# B&R Automation Studio project CombinedLinenSoiledA9KAN (part 12)

```iecst
						_PmIntern.enCycImpState := cs_ImpRdyFault;

					ELSE

						_PmIntern.enCycImpState := cs_ImpTOC;

					END_IF

				END_IF

			cs_ImpDelDir:

				_DirDeleteEx(enable := TRUE, pDevice := ADR(KG_DEVICE_COMPACTFLASH), pName := ADR(_PmIntern.sActPath));

				IF _DirDeleteEx.status <> ERR_FUB_BUSY THEN

					_PmIntern.enCycImpState := cs_ImpTOC;

				END_IF

			cs_ImpTOC:

				_PmIntern.ExpSettings.sCfDeviceName := KG_DEVICE_COMPACTFLASH;
				_PmIntern.ExpSettings.sPath := MNPARAM_PATH_EXPORT;

				_ExportTableOfContent(Enable := TRUE, pIntern := ADR(_PmIntern));

				IF _ExportTableOfContent.Status = ERR_OK THEN

					mnParamStatAd.dtExportContent := _ExportTableOfContent.dtTocWritten;

					_PmIntern.enCycImpState := cs_ImpRdySuccess;

				ELSIF _ExportTableOfContent.Status <> ERR_FUB_BUSY THEN

					_PmIntern.Status.wMsgClass := 10;
					_PmIntern.Status.wMsgNumber := MNPARAM_MSG_WARN_IMPORT;
					_PmIntern.Status.diMsgAttr1 := _ExportTableOfContent.Status;
					_PmIntern.Status.diMsgAttr2 := _ExportTableOfContent.AdStatus;
					_PmIntern.Status.wMsgAckLevel := 0;

					_PmIntern.enCycImpState := cs_ImpRdyFault;

				END_IF

			cs_ImpRdyFault:

			// Mit Fehler beendet

			cs_ImpRdySuccess:

				// Mit Erfolg beendet

		END_CASE

		//*********************************************************************************************
		// Statemachine zum Füllen des Editiors mit Daten
		//*********************************************************************************************

		CASE _PmIntern.enCycFillEditor OF

			cs_feIdle:

			cs_feStart:

				brsmemset(ADR(IFmnParam.Out.Edit.AttrNum), 0, SIZEOF(IFmnParam.Out.Edit.AttrNum));
				brsmemset(ADR(IFmnParam.Out.Edit.AttrStr), 0, SIZEOF(IFmnParam.Out.Edit.AttrStr));
				IFmnParam.Out.Edit.bCntNumRows := 0;
				IFmnParam.Out.Edit.bCntStrRows := 0;
				IFmnParam.Out.Edit.bContainer := 0;
				IFmnParam.Out.Edit.wContainerInstance := 0;
				IFmnParam.Out.Edit.wRowNumOffset := 0;
				IFmnParam.Out.Edit.wRowStrOffset := 0;

				brsmemset(ADR(_EditNumValues), 0, SIZEOF(_EditNumValues));
				brsmemset(ADR(_EditStrValues), 0, SIZEOF(_EditStrValues));

				IFmnParam.Out.Edit.wStatus := KG_STAT_BUSY;

				_DefineActContainer(Enable := TRUE, bContainerIdx := IFmnParam.In.Edit.bContainer, wInstanceIdx := IFmnParam.In.Edit.wContainerInstance, pIntern := ADR(_PmIntern));

				IF _DefineActContainer.Status = ERR_OK THEN

					// Container Parameter sind im gültigen Bereich und die Containerspec. ist ok

					IF (_PmIntern.TOC.TocEntry[_PmIntern.TOC.wStartIdx[IFmnParam.In.Edit.bContainer] + (IFmnParam.In.Edit.wContainerInstance - _PmIntern.ActContainer.wMinBound)].xExist
						AND _PmIntern.ActContainer.bDirect = 0)
						OR
						(_PmIntern.TOC.TocEntry[_PmIntern.TOC.wStartIdx[IFmnParam.In.Edit.bContainer]].xExist AND _PmIntern.ActContainer.bDirect = 1) THEN

						// Die Containerinstanz existiert

						_diCSVNum(enable := TRUE, pName := ADR(_PmIntern.ActContainer.sDoNameNum));

						IF _diCSVNum.status = ERR_OK THEN

							// Datenobjekt mit aktuellen numerischen Parametern wurde gefunden

							_PmIntern.CSVDataObjects.Adress.lCSVNum := _diCSVNum.pDatObjMem;
							_PmIntern.CSVDataObjects.Size.lCSVNum := _diCSVNum.len;
							_PmIntern.CSVDataObjects.Idents.lCSVNum := _diCSVNum.ident;

							_pDoContainerNum ACCESS _PmIntern.CSVDataObjects.Adress.lCSVNum;

							_PmIntern.CSVDataObjects.MaxIndex.lCSVNum := ( (_pDoContainerNum.Header.Do.lActEndPos - SIZEOF(mnParam_CsvDynHeader_typ)) / SIZEOF(_pDoContainerNum.CsvNum[1]) );

							_diCSVString(enable := TRUE, pName := ADR(_PmIntern.ActContainer.sDoNameString));

							IF _diCSVString.status = ERR_OK THEN

								// Datenobjekt mit aktuellen String Parametern wurde gefunden

								_PmIntern.CSVDataObjects.Adress.lCSVString := _diCSVString.pDatObjMem;
								_PmIntern.CSVDataObjects.Size.lCSVString := _diCSVString.len;
								_PmIntern.CSVDataObjects.Idents.lCSVString := _diCSVString.ident;

								_pDoContainerString ACCESS _PmIntern.CSVDataObjects.Adress.lCSVString;

								_PmIntern.CSVDataObjects.MaxIndex.lCSVString := ( (_pDoContainerString.Header.Do.lActEndPos - SIZEOF(mnParam_CsvDynHeader_typ)) / SIZEOF(_pDoContainerString.CsvString[1]) );

								_PmIntern.enCycFillEditor := cs_feFillEditor;

							ELSIF _diCSVString.status <> ERR_FUB_BUSY THEN

								_PmIntern.Status.wMsgClass := 10;
								_PmIntern.Status.wMsgNumber := MNPARAM_MSG_WARN_FILLEDITOR;
								_PmIntern.Status.diMsgAttr1 := MNPARAM_STAT_SYSERROR;
								_PmIntern.Status.diMsgAttr2 := 0;
								_PmIntern.Status.sMsgAttrTxt := _PmIntern.ActContainer.sDoNameString;
								_PmIntern.Status.wMsgAckLevel := 0;

								_PmIntern.enCycFillEditor := cs_feRdyFault;

							END_IF

						ELSIF _diCSVNum.status <> ERR_FUB_BUSY THEN

							_PmIntern.Status.wMsgClass := 10;
							_PmIntern.Status.wMsgNumber := MNPARAM_MSG_WARN_FILLEDITOR;
							_PmIntern.Status.diMsgAttr1 := MNPARAM_STAT_SYSERROR;
							_PmIntern.Status.diMsgAttr2 := 0;
							_PmIntern.Status.sMsgAttrTxt := _PmIntern.ActContainer.sDoNameNum;
							_PmIntern.Status.wMsgAckLevel := 0;

							_PmIntern.enCycFillEditor := cs_feRdyFault;

						END_IF

					ELSE

						_PmIntern.Status.wMsgClass := 10;
						_PmIntern.Status.wMsgNumber := MNPARAM_MSG_WARN_FILLEDITOR;
						_PmIntern.Status.diMsgAttr1 := MNPARAM_STAT_CONTINST_NOT_EXIST;
						_PmIntern.Status.diMsgAttr2 := 0;
						_PmIntern.Status.wMsgAckLevel := 0;

						_PmIntern.enCycFillEditor := cs_feRdyFault;

					END_IF

				ELSE

					_PmIntern.Status.wMsgClass := 10;
					_PmIntern.Status.wMsgNumber := MNPARAM_MSG_WARN_FILLEDITOR;
					_PmIntern.Status.diMsgAttr1 := _DefineActContainer.Status;
					_PmIntern.Status.diMsgAttr2 := 0;
					_PmIntern.Status.wMsgAckLevel := 0;

					_PmIntern.enCycFillEditor := cs_feRdyFault;

				END_IF

			cs_feFillEditor:

				IFmnParam.Out.Edit.bContainer := IFmnParam.In.Edit.bContainer;
				IFmnParam.Out.Edit.wContainerInstance := IFmnParam.In.Edit.wContainerInstance;
				IFmnParam.Out.Edit.wRowStrOffset := IFmnParam.In.Edit.wRowStrOffset;
				IFmnParam.Out.Edit.lPtrEditNumValues := ADR(_EditNumValues);
				IFmnParam.Out.Edit.lPtrEditStrValues := ADR(_EditStrValues);

				// Numerische Werte auslesen

				IF _PmIntern.CSVDataObjects.MaxIndex.lCSVNum > 0 AND IFmnParam.In.Edit.bCntNumRows > 0 THEN

					IF IFmnParam.In.Edit.bSelectModeNum = MNPARAM_SELECTMODE_LINEAR THEN

						IFmnParam.Out.Edit.wRowNumOffset := IFmnParam.In.Edit.wRowNumOffset;
						_wActRow := 1;
						_wActIdx := 1 + IFmnParam.In.Edit.wRowNumOffset;;

						REPEAT

							// Nur ausführen, wenn _wActIdx zulässig ist
							IF _wActIdx <= _PmIntern.CSVDataObjects.MaxIndex.lCSVNum THEN

								// Referenz auf Parameterbeschreibung auslesen
								_wActRefIdx := _pDoContainerNum.CsvNum[_wActIdx].wIdxNumPar;

								// Ist die Referenz zulässig, d.h. ist der Parameter im Modell definiert?
								IF _wActRefIdx <= _PmIntern.DataObjects.MaxIndex.lParamNum THEN

									// Schreib- und Leserechte ermitteln. Sie können vererbt sein!
									_GetAccessRights(Enable := TRUE, siWriteAccess := _pDoParamNum.ParamNum[_wActRefIdx].siWriteAccess,
										siReadAccess := _pDoParamNum.ParamNum[_wActRefIdx].siVisibleAccess,
										wReference := _pDoParamNum.ParamNum[_wActRefIdx].wReferenz,
										lPtrLogicStruct := _PmIntern.DataObjects.Adress.lLogicalStruct,
										wMaxIdxLogicStruct := UDINT_TO_UINT(_PmIntern.DataObjects.MaxIndex.lLogicalStruct));

									IF _GetAccessRights.bReadAccess <= IFmnParam.In.Edit.bUserLevel THEN

										IFmnParam.Out.Edit.AttrNum[_wActRow].bReadAccess := _GetAccessRights.bReadAccess;
										IFmnParam.Out.Edit.AttrNum[_wActRow].bWriteAccess := _GetAccessRights.bWriteAccess;

										// ***************ACTION***************
										_actFillEditNum;
										// ***************ACTION***************

										IFmnParam.Out.Edit.bCntNumRows := UINT_TO_USINT(_wActRow);

										_wActRow := _wActRow + 1;

									END_IF

								END_IF

							END_IF

							_wActIdx := _wActIdx + 1;

							UNTIL

							_PmIntern.CSVDataObjects.MaxIndex.lCSVNum < _wActIdx OR _wActRow > MIN(MNPARAM_CNT_EDITROWS, IFmnParam.In.Edit.bCntNumRows)

						END_REPEAT

					// Stringwerte auslesen, wenn gefordert

					ELSIF IFmnParam.In.Edit.bSelectModeNum = MNPARAM_SELECTMODE_BYIDX THEN

						IFmnParam.Out.Edit.wRowNumOffset := 0;
						IFmnParam.Out.Edit.bCntNumRows := UINT_TO_USINT(MIN(MNPARAM_CNT_EDITROWS, IFmnParam.In.Edit.bCntNumRows));

						FOR _ii := 1 TO IFmnParam.Out.Edit.bCntNumRows DO

							_wActRow := _ii;

							// Ist die Referenz zulässig, d.h. ist der Parameter im Modell definiert?
							IF IFmnParam.In.Edit.wSelParIdxNum[_wActRow] <= _PmIntern.DataObjects.MaxIndex.lParamNum AND IFmnParam.In.Edit.wSelParIdxNum[_wActRow] > 0 THEN

								_wActRefIdx := IFmnParam.In.Edit.wSelParIdxNum[_wActRow];

								// Suche Parameter-Containerindex anhand des Parameterindex und der 4 möglichen Array-Werte
								_binarySearchNum.enable := TRUE;
								_binarySearchNum.CsvStructNum.wIdxNumPar 	:= IFmnParam.In.Edit.wSelParIdxNum[_wActRow];
								_binarySearchNum.CsvStructNum.wArrIdx1 		:= IFmnParam.In.Edit.wSelParArrIdxNum[_wActRow,1];
								_binarySearchNum.CsvStructNum.wArrIdx2 		:= IFmnParam.In.Edit.wSelParArrIdxNum[_wActRow,2];
								_binarySearchNum.CsvStructNum.wArrIdx3 		:= IFmnParam.In.Edit.wSelParArrIdxNum[_wActRow,3];
								_binarySearchNum.CsvStructNum.wArrIdx4 		:= IFmnParam.In.Edit.wSelParArrIdxNum[_wActRow,4];
								_binarySearchNum.lpList 					:= _PmIntern.CSVDataObjects.Adress.lCSVNum;
								_binarySearchNum.lMaxRow 					:= _PmIntern.CSVDataObjects.MaxIndex.lCSVNum;

								_binarySearchNum();

								// Wurde der Parameter im Container gefunden ?
								IF _binarySearchNum.status = ERR_OK THEN

									_wActIdx := UDINT_TO_UINT(_binarySearchNum.lFoundRow);

									// Schreib- und Leserechte ermitteln. Sie können vererbt sein!
									_GetAccessRights(Enable := TRUE, siWriteAccess := _pDoParamNum.ParamNum[_wActRefIdx].siWriteAccess,
										siReadAccess := _pDoParamNum.ParamNum[_wActRefIdx].siVisibleAccess,
										wReference := _pDoParamNum.ParamNum[_wActRefIdx].wReferenz,
										lPtrLogicStruct := _PmIntern.DataObjects.Adress.lLogicalStruct,
										wMaxIdxLogicStruct := UDINT_TO_UINT(_PmIntern.DataObjects.MaxIndex.lLogicalStruct));

									IF _GetAccessRights.bReadAccess <= IFmnParam.In.Edit.bUserLevel THEN

										IFmnParam.Out.Edit.AttrNum[_wActRow].bReadAccess := _GetAccessRights.bReadAccess;
										IFmnParam.Out.Edit.AttrNum[_wActRow].bWriteAccess := _GetAccessRights.bWriteAccess;

										// ***************ACTION***************
										_actFillEditNum;
										// ***************ACTION***************

									END_IF

								END_IF

							END_IF

						END_FOR

					END_IF

				END_IF

				IF _PmIntern.CSVDataObjects.MaxIndex.lCSVString > 0 AND IFmnParam.In.Edit.bCntStrRows > 0 THEN

					IF IFmnParam.In.Edit.bSelectModeStr = MNPARAM_SELECTMODE_LINEAR THEN

						IFmnParam.Out.Edit.wRowStrOffset := IFmnParam.In.Edit.wRowStrOffset;
						_wActRow := 1;
						_wActIdx := 1 + IFmnParam.In.Edit.wRowStrOffset;;

						REPEAT

							// Nur ausführen, wenn _wActIdx zulässig ist
							IF _wActIdx <= _PmIntern.CSVDataObjects.MaxIndex.lCSVString THEN

								// Referenz auf Parameterbeschreibung auslesen
								_wActRefIdx := _pDoContainerString.CsvString[_wActIdx].wIdxStringPar;

								// Ist die Referenz zulässig, d.h. ist der Parameter im Modell definiert?
								IF _wActRefIdx <= _PmIntern.DataObjects.MaxIndex.lParamString THEN

									// Schreib- und Leserechte ermitteln. Sie können vererbt sein!
									_GetAccessRights(Enable := TRUE, siWriteAccess := _pDoParamString.ParamString[_wActRefIdx].siWriteAccess,
									siReadAccess := _pDoParamString.ParamString[_wActRefIdx].siVisibleAccess,
									wReference := _pDoParamString.ParamString[_wActRefIdx].wReferenz,
									lPtrLogicStruct := _PmIntern.DataObjects.Adress.lLogicalStruct,
									wMaxIdxLogicStruct := UDINT_TO_UINT(_PmIntern.DataObjects.MaxIndex.lLogicalStruct));

									IF _GetAccessRights.bReadAccess <= IFmnParam.In.Edit.bUserLevel THEN

										IFmnParam.Out.Edit.AttrStr[_wActRow].bReadAccess := _GetAccessRights.bReadAccess;
										IFmnParam.Out.Edit.AttrStr[_wActRow].bWriteAccess := _GetAccessRights.bWriteAccess;

										// ***************ACTION***************
										_actFillEditStr;
										// ***************ACTION***************

										IFmnParam.Out.Edit.bCntStrRows := UINT_TO_USINT(_wActRow);

										_wActRow := _wActRow + 1;

									END_IF

								END_IF

							END_IF

							_wActIdx := _wActIdx + 1;

							UNTIL

							_PmIntern.CSVDataObjects.MaxIndex.lCSVString < _wActIdx OR _wActRow > MIN(MNPARAM_CNT_EDITROWS, IFmnParam.In.Edit.bCntStrRows)

						END_REPEAT

					ELSIF IFmnParam.In.Edit.bSelectModeStr = MNPARAM_SELECTMODE_BYIDX THEN

						IFmnParam.Out.Edit.wRowStrOffset := 0;
						IFmnParam.Out.Edit.bCntStrRows := UINT_TO_USINT(MIN(MNPARAM_CNT_EDITROWS, IFmnParam.In.Edit.bCntStrRows));

						FOR _ii := 1 TO IFmnParam.Out.Edit.bCntStrRows DO

							_wActRow := _ii;

							// Ist die Referenz zulässig, d.h. ist der Parameter im Modell definiert?
							IF IFmnParam.In.Edit.wSelParIdxStr[_wActRow] <= _PmIntern.DataObjects.MaxIndex.lParamString AND IFmnParam.In.Edit.wSelParIdxStr[_wActRow] > 0 THEN

								_wActRefIdx := IFmnParam.In.Edit.wSelParIdxStr[_wActRow];

								// Suche Parameter-Containerindex anhand des Parameterindex und der 4 möglichen Array-Werte
								_binarySearchString.enable := TRUE;
								_binarySearchString.CsvStructString.wIdxStringPar 	:= IFmnParam.In.Edit.wSelParIdxStr[_wActRow];
								_binarySearchString.CsvStructString.wArrIdx1 		:= IFmnParam.In.Edit.wSelParArrIdxStr[_wActRow,1];
								_binarySearchString.CsvStructString.wArrIdx2 		:= IFmnParam.In.Edit.wSelParArrIdxStr[_wActRow,2];
								_binarySearchString.CsvStructString.wArrIdx3 		:= IFmnParam.In.Edit.wSelParArrIdxStr[_wActRow,3];
								_binarySearchString.CsvStructString.wArrIdx4 		:= IFmnParam.In.Edit.wSelParArrIdxStr[_wActRow,4];
								_binarySearchString.lpList 							:= _PmIntern.CSVDataObjects.Adress.lCSVString;
								_binarySearchString.lMaxRow 						:= _PmIntern.CSVDataObjects.MaxIndex.lCSVString;

								_binarySearchString();

								// Wurde der Parameter im Container gefunden ?
								IF _binarySearchString.status = ERR_OK THEN

									_wActIdx := UDINT_TO_UINT(_binarySearchString.lFoundRow);

									// Schreib- und Leserechte ermitteln. Sie können vererbt sein!
									_GetAccessRights(Enable := TRUE, siWriteAccess := _pDoParamString.ParamString[_wActRefIdx].siWriteAccess,
									siReadAccess := _pDoParamString.ParamString[_wActRefIdx].siVisibleAccess,
									wReference := _pDoParamString.ParamString[_wActRefIdx].wReferenz,
									lPtrLogicStruct := _PmIntern.DataObjects.Adress.lLogicalStruct,
									wMaxIdxLogicStruct := UDINT_TO_UINT(_PmIntern.DataObjects.MaxIndex.lLogicalStruct));

									IF _GetAccessRights.bReadAccess <= IFmnParam.In.Edit.bUserLevel THEN

										IFmnParam.Out.Edit.AttrStr[_wActRow].bReadAccess := _GetAccessRights.bReadAccess;
										IFmnParam.Out.Edit.AttrStr[_wActRow].bWriteAccess := _GetAccessRights.bWriteAccess;

										// ***************ACTION***************
										_actFillEditStr;
										// ***************ACTION***************

									END_IF

								END_IF

							END_IF

						END_FOR

					END_IF

				END_IF

				_PmIntern.enCycFillEditor := cs_feRdySuccess;

			cs_feRdyFault:

			// Mit Fehler beendet

			cs_feRdySuccess:

				// Erfolgreich beendet

		END_CASE

		//*********************************************************************************************
		// Statemachine zum Sichern der Daten des Editiors
		//*********************************************************************************************

		CASE _PmIntern.enCycSaveEditor OF

			cs_seIdle:

			cs_seStart:

				_DefineActContainer(Enable := TRUE, bContainerIdx := IFmnParam.In.Edit.bContainer, wInstanceIdx := IFmnParam.In.Edit.wContainerInstance, pIntern := ADR(_PmIntern));

				IF _DefineActContainer.Status = ERR_OK THEN

					// Container Parameter sind im gültigen Bereich und die Containerspec. ist ok

					IF 	(_PmIntern.TOC.TocEntry[_PmIntern.TOC.wStartIdx[IFmnParam.In.Edit.bContainer] + (IFmnParam.In.Edit.wContainerInstance - _PmIntern.ActContainer.wMinBound)].xExist
						AND _PmIntern.ActContainer.bDirect = 0)
						OR
						(_PmIntern.TOC.TocEntry[_PmIntern.TOC.wStartIdx[IFmnParam.In.Edit.bContainer]].xExist AND _PmIntern.ActContainer.bDirect = 1) THEN

						// Die Containerinstanz existiert

						_diCSVNum(enable := TRUE, pName := ADR(_PmIntern.ActContainer.sDoNameNum));

						IF _diCSVNum.status = ERR_OK THEN

							// Datenobjekt mit aktuellen numerischen Parametern wurde gefunden

							_PmIntern.CSVDataObjects.Adress.lCSVNum := _diCSVNum.pDatObjMem;
							_PmIntern.CSVDataObjects.Size.lCSVNum := _diCSVNum.len;
							_PmIntern.CSVDataObjects.Idents.lCSVNum := _diCSVNum.ident;

							_pDoContainerNum ACCESS _PmIntern.CSVDataObjects.Adress.lCSVNum;

							IF NOT _pDoContainerNum.Header.Container.xWriteProtected THEN

								_PmIntern.CSVDataObjects.MaxIndex.lCSVNum := ( (_pDoContainerNum.Header.Do.lActEndPos - SIZEOF(mnParam_CsvDynHeader_typ)) / SIZEOF(_pDoContainerNum.CsvNum[1]) );

								_diCSVString(enable := TRUE, pName := ADR(_PmIntern.ActContainer.sDoNameString));

								IF _diCSVString.status = ERR_OK THEN

									// Datenobjekt mit aktuellen String Parametern wurde gefunden

									_PmIntern.CSVDataObjects.Adress.lCSVString := _diCSVString.pDatObjMem;
									_PmIntern.CSVDataObjects.Size.lCSVString := _diCSVString.len;
									_PmIntern.CSVDataObjects.Idents.lCSVString := _diCSVString.ident;

									_pDoContainerString ACCESS _PmIntern.CSVDataObjects.Adress.lCSVString;

									_PmIntern.CSVDataObjects.MaxIndex.lCSVString := ( (_pDoContainerString.Header.Do.lActEndPos - SIZEOF(mnParam_CsvDynHeader_typ)) / SIZEOF(_pDoContainerString.CsvString[1]) );

									IF _PmIntern.ActContainer.bDirect = 0 THEN

										_diDO(enable := TRUE, pName := ADR(_PmIntern.ActContainer.sDoName));

										IF _diDO.status = ERR_OK THEN

											_PmIntern.CSVDataObjects.Adress.lDataObjekt := _diDO.pDatObjMem;
											_PmIntern.CSVDataObjects.Size.lDataObjekt := _diDO.len;
											_PmIntern.CSVDataObjects.Idents.lDataObjekt := _diDO.ident;

											IF  (PV_xgetadr(ADR(_PmIntern.ActContainer.sStrucRoot), ADR(_lPVadress), ADR(_lPVlen)) = ERR_OK) THEN

												_PmIntern.ActContainer.lAdressStructRoot := _lPVadress;
												_PmIntern.ActContainer.lSizeStructRoot := _lPVlen;

												_PmIntern.CSVDataObjects.TempAdresses.lDataObjekt := _lPVadress;
												_PmIntern.CSVDataObjects.Size.lDataObjekt := _lPVlen;

												_PmIntern.enCycSaveEditor := cs_seReadContainer;

											ELSE

												_PmIntern.Status.wMsgClass := 10;
												_PmIntern.Status.wMsgNumber := MNPARAM_MSG_WARN_SAVEEDITOR;
												_PmIntern.Status.diMsgAttr1 := MNPARAM_STAT_SYSERROR;
												_PmIntern.Status.diMsgAttr2 := 0;
												brsstrcpy(ADR(_PmIntern.Status.sMsgAttrTxt),ADR(_PmIntern.ActContainer.sStrucRoot));
												_PmIntern.Status.wMsgAckLevel := 0;

												_PmIntern.enCycSaveEditor := cs_seRdyFault;

											END_IF

										ELSIF _diDO.status <> ERR_FUB_BUSY THEN

											_PmIntern.Status.wMsgClass := 10;
											_PmIntern.Status.wMsgNumber := MNPARAM_MSG_WARN_SAVEEDITOR;
											_PmIntern.Status.diMsgAttr1 := MNPARAM_STAT_SYSERROR;
											_PmIntern.Status.diMsgAttr2 := 0;
											brsstrcpy(ADR(_PmIntern.Status.sMsgAttrTxt),ADR(_PmIntern.ActContainer.sDoName));
											_PmIntern.Status.wMsgAckLevel := 0;

											_PmIntern.enCycSaveEditor := cs_seRdyFault;

										END_IF

									ELSE

										_PmIntern.enCycSaveEditor := cs_seReadContainer;

									END_IF

								ELSIF _diCSVString.status <> ERR_FUB_BUSY THEN

									_PmIntern.Status.wMsgClass := 10;
									_PmIntern.Status.wMsgNumber := MNPARAM_MSG_WARN_SAVEEDITOR;
									_PmIntern.Status.diMsgAttr1 := MNPARAM_STAT_SYSERROR;
									_PmIntern.Status.diMsgAttr2 := 0;
									_PmIntern.Status.sMsgAttrTxt := _PmIntern.ActContainer.sDoNameString;
									_PmIntern.Status.wMsgAckLevel := 0;

									_PmIntern.enCycSaveEditor := cs_seRdyFault;

								END_IF

							ELSE

								_PmIntern.Status.wMsgClass := 10;
								_PmIntern.Status.wMsgNumber := MNPARAM_MSG_WARN_SAVEEDITOR;
								_PmIntern.Status.diMsgAttr1 := MNPARAM_STAT_WRITEPROTECTED;
								_PmIntern.Status.diMsgAttr2 := 0;
								_PmIntern.Status.sMsgAttrTxt := _PmIntern.ActContainer.sDoNameNum;
								_PmIntern.Status.wMsgAckLevel := 0;

								_PmIntern.enCycSaveEditor := cs_seRdyFault;

							END_IF

						ELSIF _diCSVNum.status <> ERR_FUB_BUSY THEN

							_PmIntern.Status.wMsgClass := 10;
							_PmIntern.Status.wMsgNumber := MNPARAM_MSG_WARN_SAVEEDITOR;
							_PmIntern.Status.diMsgAttr1 := MNPARAM_STAT_SYSERROR;
							_PmIntern.Status.diMsgAttr2 := 0;
							_PmIntern.Status.sMsgAttrTxt := _PmIntern.ActContainer.sDoNameNum;
							_PmIntern.Status.wMsgAckLevel := 0;

							_PmIntern.enCycSaveEditor := cs_seRdyFault;

						END_IF

					ELSE

						_PmIntern.Status.wMsgClass := 10;
						_PmIntern.Status.wMsgNumber := MNPARAM_MSG_WARN_SAVEEDITOR;
						_PmIntern.Status.diMsgAttr2 := 0;
						_PmIntern.Status.wMsgAckLevel := 0;

						_PmIntern.Status.diMsgAttr1 := MNPARAM_STAT_CONTINST_NOT_EXIST;

						_PmIntern.enCycSaveEditor := cs_seRdyFault;

					END_IF

				ELSE

					_PmIntern.Status.wMsgClass := 10;
					_PmIntern.Status.wMsgNumber := MNPARAM_MSG_WARN_SAVEEDITOR;
					_PmIntern.Status.diMsgAttr1 := _DefineActContainer.Status;
					_PmIntern.Status.diMsgAttr2 := 0;
					_PmIntern.Status.wMsgAckLevel := 0;

					_PmIntern.enCycSaveEditor := cs_seRdyFault;

				END_IF

			cs_seReadContainer:
			// Daten in den temporären Speicher laden

				_MemPartAlloc(enable := TRUE, ident := _MemPartCreate.ident, len := _PmIntern.CSVDataObjects.Size.lCSVNum);

				IF _MemPartAlloc.status = ERR_OK THEN

					_PmIntern.CSVDataObjects.TempAdresses.lCSVNum := _MemPartAlloc.mem;

					_drCSVNum(enable := TRUE, ident := _PmIntern.CSVDataObjects.Idents.lCSVNum, Offset := 0, pDestination := _PmIntern.CSVDataObjects.TempAdresses.lCSVNum, len := _PmIntern.CSVDataObjects.Size.lCSVNum);

					IF _drCSVNum.status = ERR_OK THEN

						_pDoContainerNum ACCESS _PmIntern.CSVDataObjects.TempAdresses.lCSVNum;

						_MemPartAlloc(enable := TRUE, ident := _MemPartCreate.ident, len := _PmIntern.CSVDataObjects.Size.lCSVString);

						IF _MemPartAlloc.status = ERR_OK THEN

							_PmIntern.CSVDataObjects.TempAdresses.lCSVString := _MemPartAlloc.mem;

							_drCSVString(enable := TRUE, ident := _PmIntern.CSVDataObjects.Idents.lCSVString, Offset := 0, pDestination := _PmIntern.CSVDataObjects.TempAdresses.lCSVString, len := _PmIntern.CSVDataObjects.Size.lCSVString);

							IF _drCSVString.status = ERR_OK THEN

								_pDoContainerString ACCESS _PmIntern.CSVDataObjects.TempAdresses.lCSVString;

								IF _PmIntern.ActContainer.bDirect  = 1 THEN

									_PmIntern.enCycSaveEditor := cs_seCommit;

								ELSE

									_drDO(enable := TRUE, ident := _PmIntern.CSVDataObjects.Idents.lDataObjekt, Offset := 0, pDestination := _PmIntern.CSVDataObjects.TempAdresses.lDataObjekt, len := _PmIntern.CSVDataObjects.Size.lDataObjekt);

									IF _drDO.status = ERR_OK THEN

										_PmIntern.enCycSaveEditor := cs_seCommit;

									ELSE

										_PmIntern.Status.wMsgClass := 10;
										_PmIntern.Status.wMsgNumber := MNPARAM_MSG_WARN_SAVEEDITOR;
										_PmIntern.Status.diMsgAttr1 := MNPARAM_STAT_IMPREADBIN;
										_PmIntern.Status.diMsgAttr2 := 0;
										_PmIntern.Status.wMsgAckLevel := 0;

										_MemPartFree(enable := TRUE, ident := _MemPartCreate.ident, mem := _PmIntern.CSVDataObjects.TempAdresses.lCSVNum);
										_MemPartFree(enable := TRUE, ident := _MemPartCreate.ident, mem := _PmIntern.CSVDataObjects.TempAdresses.lCSVString);

										_PmIntern.enCycSaveEditor := cs_seRdyFault;

									END_IF

								END_IF

							ELSE

								_PmIntern.Status.wMsgClass := 10;
								_PmIntern.Status.wMsgNumber := MNPARAM_MSG_WARN_SAVEEDITOR;
								_PmIntern.Status.diMsgAttr1 := MNPARAM_STAT_IMPREADSTR;
								_PmIntern.Status.diMsgAttr2 := 0;
								_PmIntern.Status.wMsgAckLevel := 0;

								_MemPartFree(enable := TRUE, ident := _MemPartCreate.ident, mem := _PmIntern.CSVDataObjects.TempAdresses.lCSVNum);
								_MemPartFree(enable := TRUE, ident := _MemPartCreate.ident, mem := _PmIntern.CSVDataObjects.TempAdresses.lCSVString);

								_PmIntern.enCycSaveEditor := cs_seRdyFault;

							END_IF

						ELSE

							_PmIntern.Status.wMsgClass := 10;
							_PmIntern.Status.wMsgNumber := MNPARAM_MSG_WARN_SAVEEDITOR;
							_PmIntern.Status.diMsgAttr1 := MNPARAM_STAT_IMPALLOCMEMS;
							_PmIntern.Status.diMsgAttr2 := 0;
							_PmIntern.Status.wMsgAckLevel := 0;

							_MemPartFree(enable := TRUE, ident := _MemPartCreate.ident, mem := _PmIntern.CSVDataObjects.TempAdresses.lCSVNum);

							_PmIntern.enCycSaveEditor := cs_seRdyFault;

						END_IF

					ELSE

						_PmIntern.Status.wMsgClass := 10;
						_PmIntern.Status.wMsgNumber := MNPARAM_MSG_WARN_SAVEEDITOR;
						_PmIntern.Status.diMsgAttr1 := MNPARAM_STAT_IMPREADNUM;
						_PmIntern.Status.diMsgAttr2 := 0;
						_PmIntern.Status.wMsgAckLevel := 0;

						_PmIntern.enCycSaveEditor := cs_seRdyFault;

					END_IF

				ELSE

					_PmIntern.Status.wMsgClass := 10;
					_PmIntern.Status.wMsgNumber := MNPARAM_MSG_WARN_SAVEEDITOR;
					_PmIntern.Status.diMsgAttr1 := MNPARAM_STAT_IMPALLOCMEMN;
					_PmIntern.Status.diMsgAttr2 := 0;
					_PmIntern.Status.wMsgAckLevel := 0;

					_PmIntern.enCycSaveEditor := cs_seRdyFault;

				END_IF

			cs_seCommit:

			// Daten in die Datenobjekte schreiben

				_binarySearchNum.enable := TRUE;
				_binarySearchNum.lpList := _PmIntern.CSVDataObjects.TempAdresses.lCSVNum;
				_binarySearchNum.lMaxRow := _PmIntern.CSVDataObjects.MaxIndex.lCSVNum;

				_binarySearchString.enable := TRUE;
				_binarySearchString.lpList := _PmIntern.CSVDataObjects.TempAdresses.lCSVString;
				_binarySearchString.lMaxRow := _PmIntern.CSVDataObjects.MaxIndex.lCSVString;

				_xNumDirty := FALSE;

				IF _PmIntern.CSVDataObjects.MaxIndex.lCSVNum > 0 AND IFmnParam.In.Edit.bCntNumRows > 0 AND IFmnParam.In.Edit.bCntNumRows <= MNPARAM_CNT_EDITROWS THEN

					FOR _i := 1 TO IFmnParam.Out.Edit.bCntNumRows DO

						IF _EditNumValues.xSave[_i] THEN

							_xNumDirty := TRUE;

						END_IF

					END_FOR

					IF _xNumDirty THEN

						FOR _i := 1 TO IFmnParam.Out.Edit.bCntNumRows DO

							_wActRow := _i;
							_wActIdx := _EditNumValues.wIdx[_i];

							IF _wActIdx > 0 AND _wActIdx <= _PmIntern.CSVDataObjects.MaxIndex.lCSVNum AND _EditNumValues.xSave[_wActRow] THEN

								_wActRefIdx := _pDoContainerNum.CsvNum[_wActIdx].wIdxNumPar;

								// Ist die Referenz zulässig, d.h. ist der Parameter im Modell definiert?
								IF _wActRefIdx <= _PmIntern.DataObjects.MaxIndex.lParamNum THEN

									IF _pDoParamNum.ParamNum[_wActRefIdx].bRowType = 0 THEN
										_rValue := kgUnitconfDisplayToREAL(_EditNumValues.rVal[_wActRow], _pDoParamNum.ParamNum[_wActRefIdx].wUnitID,IFmnParam.In.Edit.bLocUnit);
										_pDoContainerNum.CsvNum[_wActIdx].diValue := LIMIT(_pDoParamNum.ParamNum[_wActRefIdx].diMinValue, REAL_TO_DINT(_rValue), _pDoParamNum.ParamNum[_wActRefIdx].diMaxValue);
									ELSE
										_prMinValue ACCESS ADR(_pDoParamNum.ParamNum[_wActRefIdx].diMinValue);
										_prMaxValue ACCESS ADR(_pDoParamNum.ParamNum[_wActRefIdx].diMaxValue);
										_rValue := LIMIT(_prMinValue,kgUnitconfDisplayToREAL(_EditNumValues.rVal[_wActRow], _pDoParamNum.ParamNum[_wActRefIdx].wUnitID,IFmnParam.In.Edit.bLocUnit),_prMaxValue);
										_prValue ACCESS ADR(_pDoContainerNum.CsvNum[_wActIdx].diValue);
										_prValue := _rValue;
									END_IF

									_pDoContainerNum.CsvNum[_wActIdx].xChanged := _pDoParamNum.ParamNum[_wActRefIdx].diDefValue <> _pDoContainerNum.CsvNum[_wActIdx].diValue;

									_PN := _pDoParamNum.ParamNum[_wActRefIdx];
									_CN := _pDoContainerNum.CsvNum[_wActIdx];

									GetArrayPV(pPV := ADR(_PN.sAdresse), pStructRoot := ADR(_PmIntern.ActContainer.sStrucRoot), pPVFilled := ADR(_sPVAdress), idx1 :=_CN.wArrIdx1, idx2:=_CN.wArrIdx2, idx3:=_CN.wArrIdx3, idx4:=_CN.wArrIdx4);

									IF _CN.bRowType = 0 THEN

										_WritePVNum(pAdress := ADR(_sPVAdress), diValue := _CN.diValue);

									ELSE

										_prValue ACCESS ADR(_CN.diValue);
										_WritePVrNum(pAdress := ADR(_sPVAdress), rValue := _prValue);

									END_IF

								END_IF

								_EditNumValues.xSave[_wActRow] := FALSE;

							END_IF

						END_FOR

					END_IF

				END_IF

				IF _PmIntern.CSVDataObjects.MaxIndex.lCSVString > 0 AND IFmnParam.In.Edit.bCntStrRows > 0 AND IFmnParam.In.Edit.bCntNumRows <= MNPARAM_CNT_EDITROWS THEN

					_xStrDirty := FALSE;

					FOR _i := 1 TO IFmnParam.Out.Edit.bCntStrRows DO

						IF _EditStrValues.xSave[_i] THEN

							_xStrDirty := TRUE;

						END_IF

					END_FOR

					IF _xStrDirty THEN

						FOR _i := 1 TO IFmnParam.Out.Edit.bCntStrRows DO

							_wActRow := _i;
							_wActIdx := _EditStrValues.wIdx[_i];

							IF _wActIdx > 0 AND _wActIdx <= _PmIntern.CSVDataObjects.MaxIndex.lCSVString AND _EditStrValues.xSave[_wActRow] THEN

								_wActRefIdx := _pDoContainerString.CsvString[_wActIdx].wIdxStringPar;

								// Ist die Referenz zulässig, d.h. ist der Parameter im Modell definiert?
								IF _wActRefIdx <= _PmIntern.DataObjects.MaxIndex.lParamString THEN

									_pDoContainerString.CsvString[_wActIdx].utfValue := _EditStrValues.utfVal[_wActRow];
									_pDoContainerString.CsvString[_wActIdx].xChanged := brwcscmp(ADR(_pDoParamString.ParamString[_wActRefIdx].utfDefValue),ADR(_pDoContainerString.CsvString[_wActIdx].utfValue)) <> 0;

									_PS := _pDoParamString.ParamString[_wActRefIdx];
									_CS := _pDoContainerString.CsvString[_wActIdx];

									GetArrayPV(pPV := ADR(_PS.sAdresse), pStructRoot := ADR(_PmIntern.ActContainer.sStrucRoot), pPVFilled := ADR(_sPVAdress), idx1 :=_CS.wArrIdx1, idx2:=_CS.wArrIdx2, idx3:=_CS.wArrIdx3, idx4:=_CS.wArrIdx4);

									IF _wActRefIdx = MNPARAM_PARIDX_MACHINENAME AND ABS(_PmIntern.ActContainer.siContainerID) = MNPARAM_IDX_MACHINENAMECONTAINER THEN
										mnParamStatAd.utfMachineName := _CS.utfValue;
									END_IF

									_WritePVString(pAdress := ADR(_sPVAdress), p_utfValue := ADR(_CS.utfValue));

								END_IF

								_EditStrValues.xSave[_wActRow] := FALSE;

							END_IF

						END_FOR

					END_IF

				END_IF

				IF _xNumDirty OR _xStrDirty THEN

					_DTGetTime(enable := TRUE);

					_pDoContainerNum.Header.Time.dtTimestamp := _DTGetTime.DT1;
					_pDoContainerString.Header.Time.dtTimestamp := _DTGetTime.DT1;

					IF _PmIntern.ActContainer.bDirect = 0 THEN

						_PmIntern.enCycSaveEditor := cs_seWriteDoBin;

					ELSE

						_PmIntern.enCycSaveEditor := cs_seWriteDoNum;

					END_IF

				ELSE

					_PmIntern.enCycSaveEditor := cs_seFreeMem;

				END_IF

			cs_seWriteDoBin:

				_dwDO(enable := TRUE, ident := _PmIntern.CSVDataObjects.Idents.lDataObjekt, Offset := 0, pSource := _PmIntern.CSVDataObjects.TempAdresses.lDataObjekt, len := _PmIntern.CSVDataObjects.Size.lDataObjekt);

				IF _dwDO.status = ERR_OK THEN

					_PmIntern.enCycSaveEditor := cs_seWriteDoNum;

				ELSIF _dwDO.status <> ERR_FUB_BUSY THEN

					_PmIntern.Status.wMsgClass := MNMSG_CLASS_WARNING;
					_PmIntern.Status.wMsgNumber := MNPARAM_MSG_WARN_SAVEEDITOR;
					_PmIntern.Status.diMsgAttr1 := MNPARAM_STAT_IMPWRITEBIN;
					_PmIntern.Status.diMsgAttr2 := 0;
					_PmIntern.Status.wMsgAckLevel := 0;

					_PmIntern.enCycSaveEditor := cs_seFreeMem;

				END_IF

			cs_seWriteDoNum:

				_dwCSVNum(enable := TRUE, ident := _PmIntern.CSVDataObjects.Idents.lCSVNum, Offset := 0, pSource := _PmIntern.CSVDataObjects.TempAdresses.lCSVNum, len := _PmIntern.CSVDataObjects.Size.lCSVNum);

				IF _dwCSVNum.status = ERR_OK THEN

					_PmIntern.enCycSaveEditor := cs_seWriteDoString;
					_pDoContainerNum ACCESS _PmIntern.CSVDataObjects.Adress.lCSVNum;

				ELSIF _dwCSVNum.status <> ERR_FUB_BUSY THEN

					_PmIntern.Status.wMsgClass := MNMSG_CLASS_WARNING;
					_PmIntern.Status.wMsgNumber := MNPARAM_MSG_WARN_SAVEEDITOR;
					_PmIntern.Status.diMsgAttr1 := MNPARAM_STAT_IMPWRITENUM;
					_PmIntern.Status.diMsgAttr2 := 0;
					_PmIntern.Status.wMsgAckLevel := 0;

					_PmIntern.enCycSaveEditor := cs_seFreeMem;

				END_IF

			cs_seWriteDoString:

				_dwCSVString(enable := TRUE, ident := _PmIntern.CSVDataObjects.Idents.lCSVString, Offset := 0, pSource := _PmIntern.CSVDataObjects.TempAdresses.lCSVString, len := _PmIntern.CSVDataObjects.Size.lCSVString);

				IF _dwCSVString.status = ERR_OK THEN

					_PmIntern.enCycSaveEditor := cs_seFreeMem;
					_pDoContainerString ACCESS _PmIntern.CSVDataObjects.Adress.lCSVString;

				ELSIF _dwCSVString.status <> ERR_FUB_BUSY THEN

					_PmIntern.Status.wMsgClass := MNMSG_CLASS_WARNING;
					_PmIntern.Status.wMsgNumber := MNPARAM_MSG_WARN_SAVEEDITOR;
					_PmIntern.Status.diMsgAttr1 := MNPARAM_STAT_IMPWRITESTR;
					_PmIntern.Status.diMsgAttr2 := 0;
					_PmIntern.Status.wMsgAckLevel := 0;

					_PmIntern.enCycSaveEditor := cs_seFreeMem;

				END_IF

			cs_seFreeMem:

				IF _PmIntern.CSVDataObjects.TempAdresses.lCSVNum <> 0 THEN

					_MemPartFree(enable := TRUE, ident  := _MemPartCreate.ident, mem := _PmIntern.CSVDataObjects.TempAdresses.lCSVNum);
					_PmIntern.CSVDataObjects.TempAdresses.lCSVNum := 0;

					IF _MemPartFree.status <> ERR_OK AND _PmIntern.Status.wMsgNumber = 0 THEN

						_PmIntern.Status.wMsgClass := MNMSG_CLASS_WARNING;
						_PmIntern.Status.wMsgNumber := MNPARAM_MSG_WARN_SAVEEDITOR;
						_PmIntern.Status.diMsgAttr1 := MNPARAM_STAT_FREEMEM;
						_PmIntern.Status.diMsgAttr2 := _MemPartFree.status;
						_PmIntern.Status.wMsgAckLevel := 0;

					END_IF

				END_IF

				IF _PmIntern.CSVDataObjects.TempAdresses.lCSVString <> 0 THEN

					_MemPartFree(enable := TRUE, ident  := _MemPartCreate.ident, mem := _PmIntern.CSVDataObjects.TempAdresses.lCSVString);
					_PmIntern.CSVDataObjects.TempAdresses.lCSVString := 0;

					IF _MemPartFree.status <> ERR_OK AND _PmIntern.Status.wMsgNumber = 0 THEN

						_PmIntern.Status.wMsgClass := MNMSG_CLASS_WARNING;
						_PmIntern.Status.wMsgNumber := MNPARAM_MSG_WARN_SAVEEDITOR;
						_PmIntern.Status.diMsgAttr1 := MNPARAM_STAT_FREEMEM;
						_PmIntern.Status.diMsgAttr2 := _MemPartFree.status;
						_PmIntern.Status.wMsgAckLevel := 0;

					END_IF

				END_IF

				IF _PmIntern.Status.wMsgNumber <> 0 THEN

					IF _PmIntern.Status.diMsgAttr1 = 0 THEN
						_PmIntern.Status.diMsgAttr1 := 59999;
					END_IF
					_PmIntern.enCycSaveEditor := cs_seRdyFault;

				ELSE

					_PmIntern.enCycSaveEditor := cs_seExpCSV;

				END_IF

			cs_seExpCSV:

				_PmIntern.ExpSettings.sCfDeviceName := KG_DEVICE_COMPACTFLASH;
				_PmIntern.ExpSettings.sPath := MNPARAM_PATH_EXPORT;
				_PmIntern.ExpSettings.sFilename := _PmIntern.ActContainer.sCsvName;

				_ec(Enable := TRUE, pIntern := ADR(_PmIntern));

				IF _ec.Status = ERR_OK THEN

					_PmIntern.enCycSaveEditor := cs_seTOC;

				ELSIF _ec.Status <> ERR_FUB_BUSY THEN

					_PmIntern.Status.wMsgClass := 10;
					_PmIntern.Status.wMsgNumber := MNPARAM_MSG_WARN_SAVEEDITOR;
					_PmIntern.Status.diMsgAttr1 := _ec.Status;
					_PmIntern.Status.diMsgAttr2 := _ec.AdStatus;
					_PmIntern.Status.wMsgAckLevel := 0;

					_PmIntern.enCycSaveEditor := cs_seRdyFault;

				END_IF

			cs_seTOC:

				_PmIntern.ExpSettings.sCfDeviceName := KG_DEVICE_COMPACTFLASH;
				_PmIntern.ExpSettings.sPath := MNPARAM_PATH_EXPORT;

				_ExportTableOfContent(Enable := TRUE, pIntern := ADR(_PmIntern));

				IF _ExportTableOfContent.Status = ERR_OK THEN

					mnParamStatAd.dtExportContent := _ExportTableOfContent.dtTocWritten;

					_PmIntern.enCycSaveEditor := cs_seRdySuccess;

				ELSIF _ExportTableOfContent.Status <> ERR_FUB_BUSY THEN

					_PmIntern.Status.wMsgClass := 10;
					_PmIntern.Status.wMsgNumber := MNPARAM_MSG_WARN_SAVEEDITOR;
					_PmIntern.Status.diMsgAttr1 := _ExportTableOfContent.Status;
					_PmIntern.Status.diMsgAttr2 := _ExportTableOfContent.AdStatus;
					_PmIntern.Status.wMsgAckLevel := 0;

					_PmIntern.enCycSaveEditor := cs_seRdyFault;

				END_IF

			cs_seRdyFault:

			// Mit Fehler beendet

			cs_seRdySuccess:

				// Erfolgreich beendet

		END_CASE

		// ===========================
		// Logging
		// ===========================

		IF _xRBReady THEN

			CASE _wLogStep OF

				0:
					_ReadRB(wPtrRead := _wPtrRBread, wPtrStart := _wPtrRBstart, wPtrWrite := _wPtrRBwrite);

					IF _ReadRB.wStatus = ERR_OK THEN

						CASE _LogEntry.wErrorNo OF

							0:
								_PmIntern.Logger.text := 'OK';

							_MNPARAM_LOG_STARTIMPORT:

								IF _LogEntry.lAttr2 = MNPARAM_IMPORT_DIFFERENCE THEN
									_PmIntern.Logger.text := 'Start Import from {##AttrVar1}';
								ELSE
									_PmIntern.Logger.text := 'Start Restore from {##AttrVar1}';
								END_IF

								_PmIntern.Logger.var1 := _LogEntry.lAttr1;

							_MNPARAM_LOG_STARTDELETE:

								_PmIntern.Logger.text := 'Start Delete Container {##AttrVar1}, Instance {##AttrVar2}';
								_PmIntern.Logger.var1 := _LogEntry.lAttr1;
								_PmIntern.Logger.var2 := _LogEntry.lAttr2;

							_MNPARAM_LOG_ENDIMPORT_SUCC:

								_PmIntern.Logger.text := 'Restore/Import OK';

							_MNPARAM_LOG_ENDIMPORT_FAILED:

								_PmIntern.Logger.text := 'Restore/Import Failed: {##AttrVar1}';
								_PmIntern.Logger.var1 := _LogEntry.lAttr1;

							_MNPARAM_LOG_ENDDELETE_SUCC:

								_PmIntern.Logger.text := 'Delete OK';

							_MNPARAM_LOG_ENDDELETE_FAILED:

								_PmIntern.Logger.text := 'Delete Failed: {##AttrVar1}';
								_PmIntern.Logger.var1 := _LogEntry.lAttr1;

							_MNPARAM_LOG_STARTSAVE:

								_PmIntern.Logger.text := 'Start Save.';

							_MNPARAM_LOG_ENDSAVE_SUCC:

								_PmIntern.Logger.text := 'Save OK';

							_MNPARAM_LOG_ENDSAVE_FAILED:

								_PmIntern.Logger.text := 'Save Failed: {##AttrVar1}';
								_PmIntern.Logger.var1 := _LogEntry.lAttr1;

							_MNPARAM_LOG_FOUNDFILES:

								_PmIntern.Logger.text := 'Found {##AttrVar1} File(s)';
								_PmIntern.Logger.var1 := _LogEntry.lAttr1;

							_MNPARAM_LOG_FOUNDFILE:

								_PmIntern.Logger.text := 'Found Container {##AttrVar1} Index {##AttrVar2}';
								_PmIntern.Logger.var1 := _LogEntry.lAttr1;
								_PmIntern.Logger.var2 := _LogEntry.lAttr2;

							_MNPARAM_LOG_WRONGMACHINENO:

								_PmIntern.Logger.text := 'Wrong Machineno. Container {##AttrVar1} Index {##AttrVar2}';
								_PmIntern.Logger.var1 := _LogEntry.lAttr1;
								_PmIntern.Logger.var2 := _LogEntry.lAttr2;

							_MNPARAM_LOG_WRONGMACHINETYPE:

								_PmIntern.Logger.text := 'Wrong Machinetype Container {##AttrVar1} Index {##AttrVar2}';
								_PmIntern.Logger.var1 := _LogEntry.lAttr1;
								_PmIntern.Logger.var2 := _LogEntry.lAttr2;

							_MNPARAM_LOG_NOVERSION:

								_PmIntern.Logger.text := 'No Version in Container {##AttrVar1} Index {##AttrVar2}';
								_PmIntern.Logger.var1 := _LogEntry.lAttr1;
								_PmIntern.Logger.var2 := _LogEntry.lAttr2;

							_MNPARAM_LOG_CNTLINES:

								_PmIntern.Logger.text := 'Fault at counting lines Container {##AttrVar1} Index {##AttrVar2}';
								_PmIntern.Logger.var1 := _LogEntry.lAttr1;
								_PmIntern.Logger.var2 := _LogEntry.lAttr2;

							_MNPARAM_LOG_WRITEPROTECTED:

								_PmIntern.Logger.text := 'Write protected Container {##AttrVar1} Index {##AttrVar2}';
								_PmIntern.Logger.var1 := _LogEntry.lAttr1;
								_PmIntern.Logger.var2 := _LogEntry.lAttr2;

							_MNPARAM_LOG_SYSTEMFAULT:

								_PmIntern.Logger.text := 'System fault Container {##AttrVar1} Index {##AttrVar2}';
								_PmIntern.Logger.var1 := _LogEntry.lAttr1;
								_PmIntern.Logger.var2 := _LogEntry.lAttr2;

							_MNPARAM_LOG_STARTRESTORE:

								_PmIntern.Logger.text := 'Start Restore';

							_MNPARAM_LOG_STARTBACKUP:

								_PmIntern.Logger.text := 'Start Backup';

							_MNPARAM_LOG_ENDRESTORE_SUCC:

								_PmIntern.Logger.text := 'Restore OK';

							_MNPARAM_LOG_ENDRESTORE_FAILED:

								_PmIntern.Logger.text := 'Restore Failed: {##AttrVar1}';
								_PmIntern.Logger.var1 := _LogEntry.lAttr1;

							_MNPARAM_LOG_ENDBACKUP_SUCC:

								_PmIntern.Logger.text := 'Backup OK';

							_MNPARAM_LOG_ENDBACKUP_FAILED:

								_PmIntern.Logger.text := 'Backup Failed: {##AttrVar1}';
								_PmIntern.Logger.var1 := _LogEntry.lAttr1;

							_MNPARAM_LOG_STARTCREATE:

								_PmIntern.Logger.text := 'Start Create Container {##AttrVar1}, Instance {##AttrVar2}';
								_PmIntern.Logger.var1 := _LogEntry.lAttr1;
								_PmIntern.Logger.var2 := _LogEntry.lAttr2;

							_MNPARAM_LOG_ENDCREATE_SUCC:

								_PmIntern.Logger.text := 'Create OK';

							_MNPARAM_LOG_ENDCREATE_FAILED:

								_PmIntern.Logger.text := 'Create Failed: {##AttrVar1}';
								_PmIntern.Logger.var1 := _LogEntry.lAttr1;

							_MNPARAM_LOG_STARTCOPY:

								_PmIntern.Logger.text := 'Start Copy Container {##AttrVar1}, Instance {##AttrVar2}';
								_PmIntern.Logger.var1 := _LogEntry.lAttr1;
								_PmIntern.Logger.var2 := _LogEntry.lAttr2;

							_MNPARAM_LOG_ENDCOPY_SUCC:

								_PmIntern.Logger.text := 'Copy OK';

							_MNPARAM_LOG_ENDCOPY_FAILED:

								_PmIntern.Logger.text := 'Copy Failed: {##AttrVar1}';
								_PmIntern.Logger.var1 := _LogEntry.lAttr1;

							_MNPARAM_LOG_ROOTVAR:

								_PmIntern.Logger.text := 'Wrong rootvariable!';

							ELSE

								_PmIntern.Logger.text := UINT_TO_STRING(_LogEntry.wErrorNo);
								_PmIntern.Logger.text := CONCAT(_PmIntern.Logger.text, ' : {##AttrVar1} / {##AttrVar2}');
								_PmIntern.Logger.var1 := _LogEntry.lAttr1;
								_PmIntern.Logger.var2 := _LogEntry.lAttr2;

						END_CASE

						_wLogStep := 1;

					END_IF

				1:
					_PmIntern.Logger.logLevel := arlogLEVEL_INFO;
					_PmIntern.Logger();

					IF _PmIntern.Logger.status <> ERR_FUB_BUSY THEN

						_wLogStep := 0;

					END_IF

			END_CASE

		END_IF

		IFmnParam.Out.Edit.wCntFilesImportFailed := mnParamStatAd.wCntFilesImportFailed;
		IFmnParam.Out.Edit.wCntFilesImportFound := mnParamStatAd.wCntFilesImportFound;
		IFmnParam.Out.Edit.wCntFilesImportOK := mnParamStatAd.wCntFilesImportOK;

	ELSE // Parametermanager ist nicht bereit

		brsmemset(ADR(mnParamStatAd), 0 , SIZEOF(mnParamStatAd));
		brsmemset(ADR(IFmnParam.Out), 0 , SIZEOF(IFmnParam.Out));

		_PmIntern.Status.wMsgClass := 10;
		_PmIntern.Status.wMsgNumber := MNPARAM_MSG_SYSTEMERROR;
		_PmIntern.Status.diMsgAttr1 := 0;
		_PmIntern.Status.diMsgAttr2 := 0;
		_PmIntern.Status.wMsgAckLevel := 0;

	END_IF

	IF NOT IFmnTest.Out.xNoMessages THEN

		kgMsgStatus[MNPARAM_MSGSTATIDX] := _PmIntern.Status;

	END_IF

END_PROGRAM
```
